{attribute 'GeneratedUsingTerminal: EK1100-0000-0018'}
{attribute addProperty BoxType "EK1100-0000-0018"}
{attribute addProperty Id "Beckhoff_ELM3xxxEK1122Beckhoff_ELM3xxxEK1122_F4316A832A_0001_ELM3002_0000_0016ELM3002_73CCAB7A50A_0002_ELM3002_0000_0017ELM3002_73CCAB7A50A_0003_ELM3002_0000_0018ELM3002_73CCAB7A50A_0004_ELM3004_0000_0016ELM3004_7474644C72A_0005_ELM3004_0000_0017ELM3004_7474644C72A_0006_ELM3004_0000_0018ELM3004_7474644C72A_0007_ELM3004_0000_0019ELM3004_7474644C72"}
{attribute addProperty CRC "1992221544"}
{attribute addProperty Size "440"}
TYPE Beckhoff_ELM3xxx_76BEE368 EXTENDS EK1100_AB5A9467 :
STRUCT
	{attribute addProperty Name "Beckhoff_ELM3xxxEK1122"}
	{attribute addProperty PreviousPort "Beckhoff ELM3xxx : B"}
	Beckhoff_ELM3xxxEK1122 : Beckhoff_ELM3xxxEK1122_F4316A83;
	{attribute addProperty Name "A_0001_ELM3002_0000_0016"}
	{attribute addProperty PreviousPort "Beckhoff ELM3xxxEK1122 : C"}
	A_0001_ELM3002_0000_0016 : ELM3002_73CCAB7A;
	{attribute addProperty Name "A_0002_ELM3002_0000_0017"}
	{attribute addProperty PreviousPort "A_0001(ELM3002-0000-0016) : B"}
	A_0002_ELM3002_0000_0017 : ELM3002_73CCAB7A;
	{attribute addProperty Name "A_0003_ELM3002_0000_0018"}
	{attribute addProperty PreviousPort "A_0002(ELM3002-0000-0017) : B"}
	A_0003_ELM3002_0000_0018 : ELM3002_73CCAB7A;
	{attribute addProperty Name "A_0004_ELM3004_0000_0016"}
	{attribute addProperty PreviousPort "A_0003(ELM3002-0000-0018) : B"}
	A_0004_ELM3004_0000_0016 : ELM3004_7474644C;
	{attribute addProperty Name "A_0005_ELM3004_0000_0017"}
	{attribute addProperty PreviousPort "A_0004(ELM3004-0000-0016) : B"}
	A_0005_ELM3004_0000_0017 : ELM3004_7474644C;
	{attribute addProperty Name "A_0006_ELM3004_0000_0018"}
	{attribute addProperty PreviousPort "A_0005(ELM3004-0000-0017) : B"}
	A_0006_ELM3004_0000_0018 : ELM3004_7474644C;
	{attribute addProperty Name "A_0007_ELM3004_0000_0019"}
	{attribute addProperty PreviousPort "A_0006(ELM3004-0000-0018) : B"}
	A_0007_ELM3004_0000_0019 : ELM3004_7474644C;
END_STRUCT
END_TYPE

(* stored: Version 1.2.0.0, ProductVersion 3.1.4024.9
   DUT Beckhoff_ELM3xxx_76BEE368: Id {c086eaa7-274b-46d8-b790-273459b92083} *)
